(* IEC 61131-3 sources: AXOpen/src/components.rexroth.drives/app/src/IO/PLC_LINE, 4 files *)

(* ---- HwIdentifiers.st ---- *)
TYPE
    HwIdentifiers : WORD
    (
        ST3_indradrive_HwID :=	WORD#260,
        ST3_indradrive_F_Modul_not_used_ID_FMod_NotUsed_HwID :=	WORD#266,
        ST3_indradrive_Input_9_Words_ID_InMod_9Words_HwID :=	WORD#264,
        ST3_indradrive_Output_13_Words_ID_OutMod_13Words_HwID :=	WORD#263,
        ST3_indradrive_ParamCh_5Words_ID_PaCh_5Words_HwID :=	WORD#265,
        ST3_indradrive_Rack_HwID :=	WORD#261,
        ST3_indradrive_ST3_indradrive_HwID :=	WORD#262,
        ST3_indradrive_ST3_indradrive_DAP_1_HwID :=	WORD#267,
        ST3_indradrive_ST3_indradrive_profinet_HwID :=	WORD#257,
        ST3_indradrive_ST3_indradrive_profinet_Port_1_HwID :=	WORD#258,
        ST3_indradrive_ST3_indradrive_profinet_Port_2_HwID :=	WORD#259,
        plc_line_HwID :=	WORD#32,
        plc_line_Rail_0_HwID :=	WORD#268,
        plc_line_plc_line_HwID :=	WORD#48,
        plc_line_plc_line_CPU_display_1_HwID :=	WORD#54,
        plc_line_plc_line_Card_reader_writer_1_HwID :=	WORD#51,
        plc_line_plc_line_DP_interface_1_HwID :=	WORD#60,
        plc_line_plc_line_OPC_UA_1_HwID :=	WORD#117,
        plc_line_plc_line_profinet_x1_HwID :=	WORD#64,
        plc_line_plc_line_profinet_x1_Port_1_HwID :=	WORD#65,
        plc_line_plc_line_profinet_x1_Port_2_HwID :=	WORD#66,
        plc_line_plc_line_profinet_x2_HwID :=	WORD#72,
        plc_line_plc_line_profinet_x2_Port_3_HwID :=	WORD#73,
        plc_line_plc_line_virtual_communication_interface_HwID :=	WORD#135,
        profinet_plc_line_HwID :=	WORD#256,

        NONE := WORD#0
    );
END_TYPE

(* ---- HwInputs.st ---- *)
TYPE
	HwInputs : STRUCT
		ST3_indradrive_ParamCh_IDN_1 AT %B10 : ARRAY[0..9] OF BYTE;
		ST3_indradrive_Input_9_Words_1 AT %B20 : ARRAY[0..17] OF BYTE;
	END_STRUCT;
END_TYPE

(* ---- CopyInputs.st ---- *)
FUNCTION CopyInputs
	VAR_EXTERNAL
		HwInputs : HwInputs;
		PlcInputs : PlcInputs;
	END_VAR
	PlcInputs.ST3_indradrive_ParamCh_IDN_1[0] := HwInputs.ST3_indradrive_ParamCh_IDN_1[0];
	PlcInputs.ST3_indradrive_ParamCh_IDN_1[1] := HwInputs.ST3_indradrive_ParamCh_IDN_1[1];
	PlcInputs.ST3_indradrive_ParamCh_IDN_1[2] := HwInputs.ST3_indradrive_ParamCh_IDN_1[2];
	PlcInputs.ST3_indradrive_ParamCh_IDN_1[3] := HwInputs.ST3_indradrive_ParamCh_IDN_1[3];
	PlcInputs.ST3_indradrive_ParamCh_IDN_1[4] := HwInputs.ST3_indradrive_ParamCh_IDN_1[4];
	PlcInputs.ST3_indradrive_ParamCh_IDN_1[5] := HwInputs.ST3_indradrive_ParamCh_IDN_1[5];
	PlcInputs.ST3_indradrive_ParamCh_IDN_1[6] := HwInputs.ST3_indradrive_ParamCh_IDN_1[6];
	PlcInputs.ST3_indradrive_ParamCh_IDN_1[7] := HwInputs.ST3_indradrive_ParamCh_IDN_1[7];
	PlcInputs.ST3_indradrive_ParamCh_IDN_1[8] := HwInputs.ST3_indradrive_ParamCh_IDN_1[8];
	PlcInputs.ST3_indradrive_ParamCh_IDN_1[9] := HwInputs.ST3_indradrive_ParamCh_IDN_1[9];
	PlcInputs.ST3_indradrive_Input_9_Words_1[0] := HwInputs.ST3_indradrive_Input_9_Words_1[0];
	PlcInputs.ST3_indradrive_Input_9_Words_1[1] := HwInputs.ST3_indradrive_Input_9_Words_1[1];
	PlcInputs.ST3_indradrive_Input_9_Words_1[2] := HwInputs.ST3_indradrive_Input_9_Words_1[2];
	PlcInputs.ST3_indradrive_Input_9_Words_1[3] := HwInputs.ST3_indradrive_Input_9_Words_1[3];
	PlcInputs.ST3_indradrive_Input_9_Words_1[4] := HwInputs.ST3_indradrive_Input_9_Words_1[4];
	PlcInputs.ST3_indradrive_Input_9_Words_1[5] := HwInputs.ST3_indradrive_Input_9_Words_1[5];
	PlcInputs.ST3_indradrive_Input_9_Words_1[6] := HwInputs.ST3_indradrive_Input_9_Words_1[6];
	PlcInputs.ST3_indradrive_Input_9_Words_1[7] := HwInputs.ST3_indradrive_Input_9_Words_1[7];
	PlcInputs.ST3_indradrive_Input_9_Words_1[8] := HwInputs.ST3_indradrive_Input_9_Words_1[8];
	PlcInputs.ST3_indradrive_Input_9_Words_1[9] := HwInputs.ST3_indradrive_Input_9_Words_1[9];
	PlcInputs.ST3_indradrive_Input_9_Words_1[10] := HwInputs.ST3_indradrive_Input_9_Words_1[10];
	PlcInputs.ST3_indradrive_Input_9_Words_1[11] := HwInputs.ST3_indradrive_Input_9_Words_1[11];
	PlcInputs.ST3_indradrive_Input_9_Words_1[12] := HwInputs.ST3_indradrive_Input_9_Words_1[12];
	PlcInputs.ST3_indradrive_Input_9_Words_1[13] := HwInputs.ST3_indradrive_Input_9_Words_1[13];
	PlcInputs.ST3_indradrive_Input_9_Words_1[14] := HwInputs.ST3_indradrive_Input_9_Words_1[14];
	PlcInputs.ST3_indradrive_Input_9_Words_1[15] := HwInputs.ST3_indradrive_Input_9_Words_1[15];
	PlcInputs.ST3_indradrive_Input_9_Words_1[16] := HwInputs.ST3_indradrive_Input_9_Words_1[16];
	PlcInputs.ST3_indradrive_Input_9_Words_1[17] := HwInputs.ST3_indradrive_Input_9_Words_1[17];
END_FUNCTION

(* ---- CopyOutputs.st ---- *)
FUNCTION CopyOutputs
	VAR_EXTERNAL
		HwOutputs : HwOutputs;
		PlcOutputs : PlcOutputs;
	END_VAR
	HwOutputs.ST3_indradrive_ParamCh_IDN_1[0] := PlcOutputs.ST3_indradrive_ParamCh_IDN_1[0];
	HwOutputs.ST3_indradrive_ParamCh_IDN_1[1] := PlcOutputs.ST3_indradrive_ParamCh_IDN_1[1];
	HwOutputs.ST3_indradrive_ParamCh_IDN_1[2] := PlcOutputs.ST3_indradrive_ParamCh_IDN_1[2];
	HwOutputs.ST3_indradrive_ParamCh_IDN_1[3] := PlcOutputs.ST3_indradrive_ParamCh_IDN_1[3];
	HwOutputs.ST3_indradrive_ParamCh_IDN_1[4] := PlcOutputs.ST3_indradrive_ParamCh_IDN_1[4];
	HwOutputs.ST3_indradrive_ParamCh_IDN_1[5] := PlcOutputs.ST3_indradrive_ParamCh_IDN_1[5];
	HwOutputs.ST3_indradrive_ParamCh_IDN_1[6] := PlcOutputs.ST3_indradrive_ParamCh_IDN_1[6];
	HwOutputs.ST3_indradrive_ParamCh_IDN_1[7] := PlcOutputs.ST3_indradrive_ParamCh_IDN_1[7];
	HwOutputs.ST3_indradrive_ParamCh_IDN_1[8] := PlcOutputs.ST3_indradrive_ParamCh_IDN_1[8];
	HwOutputs.ST3_indradrive_ParamCh_IDN_1[9] := PlcOutputs.ST3_indradrive_ParamCh_IDN_1[9];
	HwOutputs.ST3_indradrive_Output_13_Words_1[0] := PlcOutputs.ST3_indradrive_Output_13_Words_1[0];
	HwOutputs.ST3_indradrive_Output_13_Words_1[1] := PlcOutputs.ST3_indradrive_Output_13_Words_1[1];
	HwOutputs.ST3_indradrive_Output_13_Words_1[2] := PlcOutputs.ST3_indradrive_Output_13_Words_1[2];
	HwOutputs.ST3_indradrive_Output_13_Words_1[3] := PlcOutputs.ST3_indradrive_Output_13_Words_1[3];
	HwOutputs.ST3_indradrive_Output_13_Words_1[4] := PlcOutputs.ST3_indradrive_Output_13_Words_1[4];
	HwOutputs.ST3_indradrive_Output_13_Words_1[5] := PlcOutputs.ST3_indradrive_Output_13_Words_1[5];
	HwOutputs.ST3_indradrive_Output_13_Words_1[6] := PlcOutputs.ST3_indradrive_Output_13_Words_1[6];
	HwOutputs.ST3_indradrive_Output_13_Words_1[7] := PlcOutputs.ST3_indradrive_Output_13_Words_1[7];
	HwOutputs.ST3_indradrive_Output_13_Words_1[8] := PlcOutputs.ST3_indradrive_Output_13_Words_1[8];
	HwOutputs.ST3_indradrive_Output_13_Words_1[9] := PlcOutputs.ST3_indradrive_Output_13_Words_1[9];
	HwOutputs.ST3_indradrive_Output_13_Words_1[10] := PlcOutputs.ST3_indradrive_Output_13_Words_1[10];
	HwOutputs.ST3_indradrive_Output_13_Words_1[11] := PlcOutputs.ST3_indradrive_Output_13_Words_1[11];
	HwOutputs.ST3_indradrive_Output_13_Words_1[12] := PlcOutputs.ST3_indradrive_Output_13_Words_1[12];
	HwOutputs.ST3_indradrive_Output_13_Words_1[13] := PlcOutputs.ST3_indradrive_Output_13_Words_1[13];
	HwOutputs.ST3_indradrive_Output_13_Words_1[14] := PlcOutputs.ST3_indradrive_Output_13_Words_1[14];
	HwOutputs.ST3_indradrive_Output_13_Words_1[15] := PlcOutputs.ST3_indradrive_Output_13_Words_1[15];
	HwOutputs.ST3_indradrive_Output_13_Words_1[16] := PlcOutputs.ST3_indradrive_Output_13_Words_1[16];
	HwOutputs.ST3_indradrive_Output_13_Words_1[17] := PlcOutputs.ST3_indradrive_Output_13_Words_1[17];
	HwOutputs.ST3_indradrive_Output_13_Words_1[18] := PlcOutputs.ST3_indradrive_Output_13_Words_1[18];
	HwOutputs.ST3_indradrive_Output_13_Words_1[19] := PlcOutputs.ST3_indradrive_Output_13_Words_1[19];
	HwOutputs.ST3_indradrive_Output_13_Words_1[20] := PlcOutputs.ST3_indradrive_Output_13_Words_1[20];
	HwOutputs.ST3_indradrive_Output_13_Words_1[21] := PlcOutputs.ST3_indradrive_Output_13_Words_1[21];
	HwOutputs.ST3_indradrive_Output_13_Words_1[22] := PlcOutputs.ST3_indradrive_Output_13_Words_1[22];
	HwOutputs.ST3_indradrive_Output_13_Words_1[23] := PlcOutputs.ST3_indradrive_Output_13_Words_1[23];
	HwOutputs.ST3_indradrive_Output_13_Words_1[24] := PlcOutputs.ST3_indradrive_Output_13_Words_1[24];
	HwOutputs.ST3_indradrive_Output_13_Words_1[25] := PlcOutputs.ST3_indradrive_Output_13_Words_1[25];
END_FUNCTION
